FUNCTION_BLOCK FLASHERT (* Multi-purpose LED Flasher *)
  (* Standard: 61499 ITA *)
  (* Version 0.0, 2004-01-09, JHC, Rockwell Automation, Copied from FLASHER4. *)
  (* Compiler header: package fb.rt.test; *)
  (* Compiler Java IBM VisualAge 3.0 *)
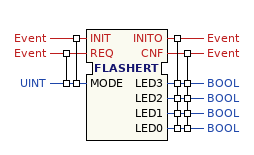
  EVENT_INPUT
    INIT WITH MODE; (* Initialization Request *)
    REQ WITH MODE; (* Update Request *)
  END_EVENT
  EVENT_OUTPUT
    INITO WITH LED3, LED2, LED1, LED0; (* Initialization Confirm *)
    CNF WITH LED3, LED2, LED1, LED0; (* Update Confirmation *)
  END_EVENT
  VAR_INPUT
    MODE : UINT; (* 0=FLASH_ALL,1=COUNT_UP,2=COUNT_DOWN,3=CHASE_UP,4=CHASE_DOWN *)
  END_VAR
  VAR_OUTPUT
    LED3 : BOOL; (* MSB *)
    LED2 : BOOL;
    LED1 : BOOL;
    LED0 : BOOL; (* LSB *)
  END_VAR
  VAR
    OFLO : BOOL;
  END_VAR
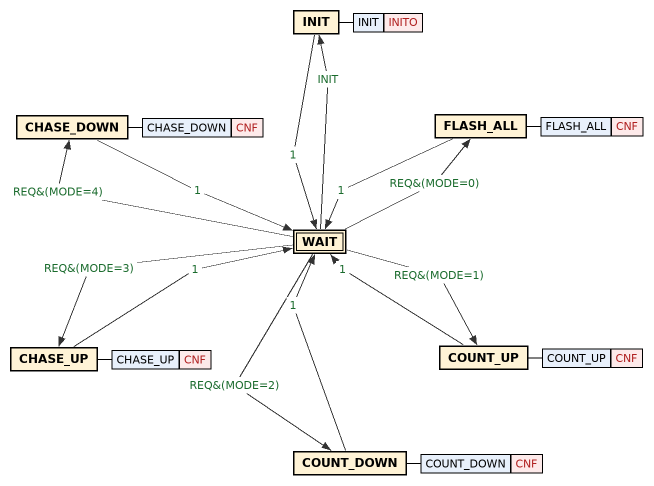
  EC_STATES
    WAIT;
    INIT : INIT -> INITO;
    FLASH_ALL : FLASH_ALL -> CNF;
    COUNT_UP : COUNT_UP -> CNF;
    COUNT_DOWN : COUNT_DOWN -> CNF;
    CHASE_UP : CHASE_UP -> CNF;
    CHASE_DOWN : CHASE_DOWN -> CNF;
  END_STATES
  EC_TRANSITIONS
    WAIT TO INIT := INIT;
    WAIT TO FLASH_ALL := REQ&(MODE=0);
    WAIT TO COUNT_UP := REQ&(MODE=1);
    WAIT TO COUNT_DOWN := REQ&(MODE=2);
    WAIT TO CHASE_UP := REQ&(MODE=3);
    WAIT TO CHASE_DOWN := REQ&(MODE=4);
    INIT TO WAIT := 1;
    FLASH_ALL TO WAIT := 1;
    COUNT_UP TO WAIT := 1;
    COUNT_DOWN TO WAIT := 1;
    CHASE_UP TO WAIT := 1;
    CHASE_DOWN TO WAIT := 1;
  END_TRANSITIONS
  ALGORITHM INIT IN ST:
LED0:=(MODE>2);
LED1:=false;
LED2:=false;
LED3:=false;
  END_ALGORITHM
  ALGORITHM COUNT_UP IN ST:
LED0:=NOT LED0;
IF NOT LED0 THEN
LED1:=NOT LED1;
IF NOT LED1 THEN
LED2:=NOT LED2;
IF NOT LED2 THEN LED3:=NOT LED3;END_IF;
END_IF;
END_IF;
  END_ALGORITHM
  ALGORITHM COUNT_DOWN IN ST:
LED0:=NOT LED0;
IF LED0 THEN
LED1:=NOT LED1;
IF LED1 THEN
LED2:=NOT LED2;
IF LED2 THEN LED3:=NOT LED3;END_IF;
END_IF;
END_IF;
  END_ALGORITHM
  ALGORITHM FLASH_ALL IN LD:
    LED0 := LED0 ! ;
    LED1 := LED1 ! ;
    LED2 := LED2 ! ;
    LED3 := LED3 ! ;
  END_ALGORITHM
  ALGORITHM CHASE_UP IN LD:
    OFLO := LED3 ;
    LED3 := LED2 ;
    LED2 := LED1 ;
    LED1 := LED0 ;
    LED0 := OFLO ;
  END_ALGORITHM
  ALGORITHM CHASE_DOWN IN LD:
    OFLO := LED0 ;
    LED0 := LED1 ;
    LED1 := LED2 ;
    LED2 := LED3 ;
    LED3 := OFLO ;
  END_ALGORITHM
END_FUNCTION_BLOCK
